TYPE
    ST_MyComponent_Status : STRUCT
        Extended   : BOOL;
        Retracted  : BOOL;
        Extending  : BOOL;
        Retracting : BOOL;
    END_STRUCT
END_TYPE

(* stored: Version 1.1.0.1
   DUT ST_MyComponent_Status: Id {49c7ec6a-2041-4957-9561-662d6c79c607} *)
